FUNCTION_BLOCK FB_Interlock
VAR_INPUT
END_VAR
VAR_OUTPUT
END_VAR
VAR
END_VAR

END_FUNCTION_BLOCK

(* stored: Version 1.1.0.1, ProductVersion 3.1.4024.12
   POU FB_Interlock: Id {0f8e4d62-4669-4071-bb6b-34004672bcd7}, SpecialFunc None *)
